// TIA Portal V17 export
// export: Created 2022-07-16T16:56:11.5436582Z, ExportSetting WithDefaults, DisplayName Totally Integrated Automation Portal, DisplayVersion V17, DisplayName TIA Portal Openness, DisplayVersion V17, DisplayName TIA Portal Version Control Interface, DisplayVersion V17, DisplayName TIA Portal Test Suite Advanced, DisplayVersion V17, DisplayName STEP 7 Professional, DisplayVersion V17, DisplayName STEP 7 Safety, DisplayVersion V17, DisplayName WinCC Professional, DisplayVersion V17
TYPE "udtSolenoidValve"
// stored: IsFailsafeCompliant false
   STRUCT
      scaledValeu : Int := 1;
      rawValue : Int := 2;
      rawMinimum : Int := 3;
      rawMaximum : Int := 4;
      scalledMinimum : Int := 5;
      scalledMaximium : Int := 6;
   END_STRUCT;
END_TYPE
